// TIA Portal project "binhtron" (V15)

(* hardware
DEVICE "S7-1200 station_1"  S7-1200 Station
   slot 0: "Rack_0"  S7-1200 Rack  Rack  V1.0
   slot 1: "PLC_1"  CPU 1212C DC/DC/DC  6ES7 212-1AE40-0XB0  V4.2
DEVICE "HMI_1"  TP1500 Comfort
   slot 0: "HMI_1"  TP1500 Comfort  6AV2 124-0QC02-0AX1  15.0.0.0
   slot 1: "HMI_RT_1"  TP1500 Comfort  6AV2 124-0QC02-0AX1  15.0.0.0
   slot 5: "HMI_1.IE_CP_1"  PROFINET Interface  15.0.0.0
      slot 1: "PROFINET Interface_1"  PROFINET Interface
         slot 1: "Port_1"  Port
         slot 2: "Port_2"  Port
   slot 6: "HMI_1.IE_CP_2"  PROFINET Interface  15.0.0.0
      slot 1: "PROFINET Interface_GBit"  PROFINET Interface
         slot 1: "Port_1"  Port
   slot 7: "HMI_1.MPI/DP_CP_1"  MPI/DP Interface  15.0.0.0
*)

// ===== PLC "PLC_1"  CPU 1212C DC/DC/DC =====

VAR_GLOBAL   // PLC tag table "Default tag table"
   "System_Byte" AT %MB1 : Byte;
   "FirstScan" AT %M1.0 : Bool;
   "DiagStatusUpdate" AT %M1.1 : Bool;
   "AlwaysTRUE" AT %M1.2 : Bool;
   "AlwaysFALSE" AT %M1.3 : Bool;
   "Clock_Byte" AT %MB0 : Byte;
   "Clock_10Hz" AT %M0.0 : Bool;
   "Clock_5Hz" AT %M0.1 : Bool;
   "Clock_2.5Hz" AT %M0.2 : Bool;
   "Clock_2Hz" AT %M0.3 : Bool;
   "Clock_1.25Hz" AT %M0.4 : Bool;
   "Clock_1Hz" AT %M0.5 : Bool;
   "Clock_0.625Hz" AT %M0.6 : Bool;
   "Clock_0.5Hz" AT %M0.7 : Bool;
   "Pump" AT %Q0.0 : Bool;
   "V" AT %Q0.1 : Bool;
END_VAR

DATA_BLOCK "DB"   // DB1
{ S7_Optimized_Access := 'FALSE' }
VERSION : 0.1
   VAR
      Auto_Man : Bool;
      Start_auto : Bool;
      Stop_auto : Bool;
      Auto : Bool;
      Pump_auto : Bool;
      V_auto : Bool;
      S1_hight : Bool;
      S2_low : Bool;
      TG : Bool;
      PV_T1 : DInt;
      PV_T2 : DInt;
      start_man_pump : Bool;
      stop_man_pump : Bool;
      pump_man : Bool;
      V_man : Bool;
      start_man_V : Bool;
      stop_man_V : Bool;
      level_water : DInt;
   END_VAR
BEGIN
END_DATA_BLOCK

// folder: System blocks/Program resources

DATA_BLOCK "IEC_Timer_0_DB"   // DB2
{ S7_Optimized_Access := 'TRUE' }
AUTHOR : Simatic
FAMILY : IEC
NAME : IEC_TMR
VERSION : 1.0
// stored: InstanceOfName IEC_TIMER
"IEC_TIMER"
BEGIN
END_DATA_BLOCK

DATA_BLOCK "T2"   // DB3
{ S7_Optimized_Access := 'TRUE' }
AUTHOR : Simatic
FAMILY : IEC
NAME : IEC_TMR
VERSION : 1.0
// stored: InstanceOfName IEC_TIMER
"IEC_TIMER"
BEGIN
END_DATA_BLOCK

DATA_BLOCK "IEC_Counter_0_DB"   // DB4
{ S7_Optimized_Access := 'TRUE' }
AUTHOR : Simatic
FAMILY : IEC
NAME : CNTR
VERSION : 1.0
// stored: InstanceOfName IEC_COUNTER
"IEC_COUNTER"
BEGIN
END_DATA_BLOCK

// folder: (top level)

FUNCTION "Auto" : Void   // FC1, LAD
{ S7_Optimized_Access := 'TRUE' }
VERSION : 0.1
   VAR_TEMP   // added for the SCL form of the ladder/FBD networks
      _w1 : Bool;
   END_VAR
BEGIN

REGION Network 1
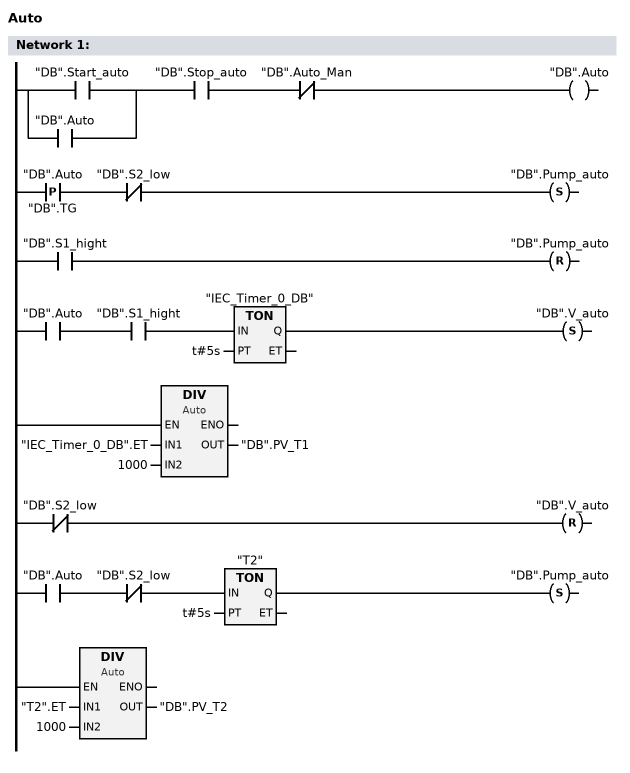
   "DB".Auto := ("DB".Start_auto OR "DB".Auto) AND "DB".Stop_auto AND NOT "DB".Auto_Man;
   #_w1 := "DB".Auto AND NOT "DB".TG;   // rising edge of "DB".Auto
   "DB".TG := "DB".Auto;
   IF #_w1 AND NOT "DB".S2_low THEN "DB".Pump_auto := TRUE; END_IF;
   IF "DB".S1_hight THEN "DB".Pump_auto := FALSE; END_IF;
   "IEC_Timer_0_DB".TON(IN := "DB".Auto AND "DB".S1_hight, PT := t#5s);
   IF "IEC_Timer_0_DB".Q THEN "DB".V_auto := TRUE; END_IF;
   "DB".PV_T1 := "IEC_Timer_0_DB".ET / 1000;
   IF NOT "DB".S2_low THEN "DB".V_auto := FALSE; END_IF;
   "T2".TON(IN := "DB".Auto AND NOT "DB".S2_low, PT := t#5s);
   IF "T2".Q THEN "DB".Pump_auto := TRUE; END_IF;
   "DB".PV_T2 := "T2".ET / 1000;
END_REGION
END_FUNCTION

FUNCTION "Man" : Void   // FC2, LAD
{ S7_Optimized_Access := 'TRUE' }
VERSION : 0.1
BEGIN

REGION Network 1
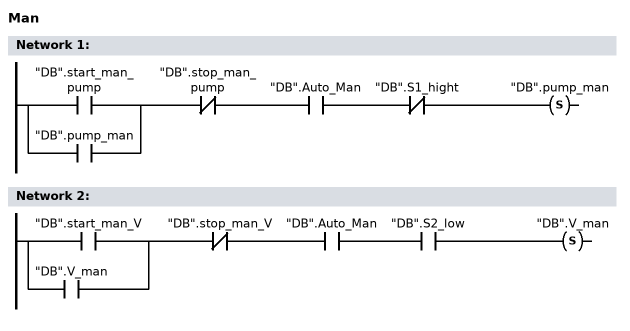
   RUNG wire#powerrail
      Contact( "DB".start_man_pump )
      wire#w1
      I_Contact( "DB".stop_man_pump )
      Contact( "DB".Auto_Man )
      I_Contact( "DB".S1_hight )
      S_Coil( "DB".pump_man )
   END_RUNG
   RUNG wire#powerrail
      Contact( "DB".pump_man )
   END_RUNG wire#w1
   // the same network as SCL:
   IF ("DB".start_man_pump OR "DB".pump_man) AND NOT "DB".stop_man_pump AND "DB".Auto_Man AND NOT "DB".S1_hight THEN
       "DB".pump_man := TRUE;
   END_IF;
END_REGION

REGION Network 2
   RUNG wire#powerrail
      Contact( "DB".start_man_V )
      wire#w1
      I_Contact( "DB".stop_man_V )
      Contact( "DB".Auto_Man )
      Contact( "DB".S2_low )
      S_Coil( "DB".V_man )
   END_RUNG
   RUNG wire#powerrail
      Contact( "DB".V_man )
   END_RUNG wire#w1
   // the same network as SCL:
   IF ("DB".start_man_V OR "DB".V_man) AND NOT "DB".stop_man_V AND "DB".Auto_Man AND "DB".S2_low THEN
       "DB".V_man := TRUE;
   END_IF;
END_REGION
END_FUNCTION

FUNCTION "Map_out" : Void   // FC3, LAD
{ S7_Optimized_Access := 'TRUE' }
VERSION : 0.1
BEGIN

REGION Network 1
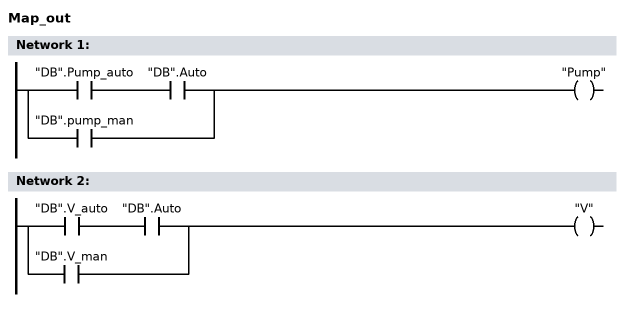
   RUNG wire#powerrail
      Contact( "DB".Pump_auto )
      Contact( "DB".Auto )
      wire#w1
      Coil( "Pump" )
   END_RUNG
   RUNG wire#powerrail
      Contact( "DB".pump_man )
   END_RUNG wire#w1
   // the same network as SCL:
   "Pump" := ("DB".Pump_auto AND "DB".Auto) OR "DB".pump_man;
END_REGION

REGION Network 2
   RUNG wire#powerrail
      Contact( "DB".V_auto )
      Contact( "DB".Auto )
      wire#w1
      Coil( "V" )
   END_RUNG
   RUNG wire#powerrail
      Contact( "DB".V_man )
   END_RUNG wire#w1
   // the same network as SCL:
   "V" := ("DB".V_auto AND "DB".Auto) OR "DB".V_man;
END_REGION
END_FUNCTION

FUNCTION "HMI_mucnuoc_sensor" : Void   // FC4, LAD
{ S7_Optimized_Access := 'TRUE' }
VERSION : 0.1
BEGIN

REGION Network 1
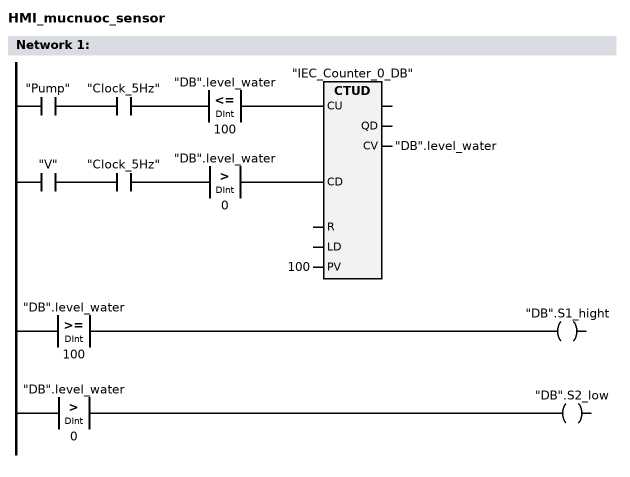
   "IEC_Counter_0_DB".CTUD(CU := "Pump" AND "Clock_5Hz" AND ("DB".level_water <= 100),
                           CD := "V" AND "Clock_5Hz" AND ("DB".level_water > 0),
                           PV := 100,
                           CV => "DB".level_water);
   "DB".S1_hight := "DB".level_water >= 100;
   "DB".S2_low := "DB".level_water > 0;
END_REGION
END_FUNCTION

ORGANIZATION_BLOCK "Main"   // OB1, LAD, ProgramCycle
TITLE = "Main Program Sweep (Cycle)"
{ S7_Optimized_Access := 'TRUE' }
VERSION : 0.1
   VAR_INPUT
      Initial_Call : Bool;   // Initial call of this OB
      Remanence : Bool;   // =True, if remanent data are available
   END_VAR
BEGIN

REGION Network 1
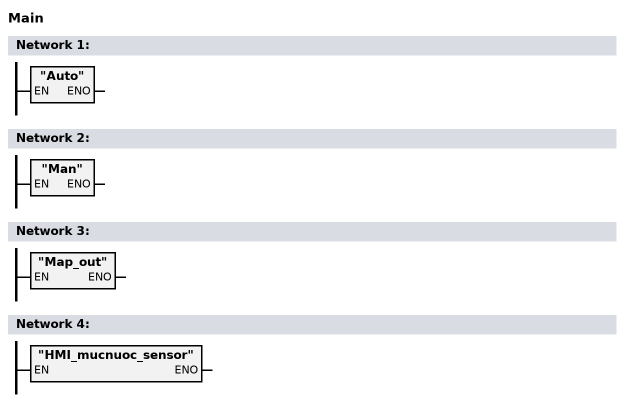
   RUNG wire#powerrail
      "Auto"()
   END_RUNG
   // the same network as SCL:
   "Auto"();
END_REGION

REGION Network 2
   RUNG wire#powerrail
      "Man"()
   END_RUNG
   // the same network as SCL:
   "Man"();
END_REGION

REGION Network 3
   RUNG wire#powerrail
      "Map_out"()
   END_RUNG
   // the same network as SCL:
   "Map_out"();
END_REGION

REGION Network 4
   RUNG wire#powerrail
      "HMI_mucnuoc_sensor"()
   END_RUNG
   // the same network as SCL:
   "HMI_mucnuoc_sensor"();
END_REGION
END_ORGANIZATION_BLOCK

(* ===== HMI "HMI_RT_1" =====
system functions are stored by id; their names below are inferred from use
connection "HMI_Connection_1": ETHERNET, S7_1200_OMS

HMI tags "Default tag table"
   "DB_Auto_Man" : Bool = PLC "DB".Auto_Man AT %DB1.DBX0.0, 1 s
   "DB_Start_auto" : Bool = PLC "DB".Start_auto AT %DB1.DBX0.1, 1 s
   "DB_Stop_auto" : Bool = PLC "DB".Stop_auto AT %DB1.DBX0.2, 1 s
   "Pump" : Bool = PLC Pump AT %Q0.0, 1 s
   "DB_level_water" : DInt = PLC "DB".level_water AT %DB1.DBD12, 1 s
   "V" : Bool = PLC V AT %Q0.1, 1 s
   "DB_S1_hight" : Bool = PLC "DB".S1_hight AT %DB1.DBX0.6, 1 s
   "DB_S2_low" : Bool = PLC "DB".S2_low AT %DB1.DBX0.7, 1 s
   "DB_PV_T1" : DInt = PLC "DB".PV_T1 AT %DB1.DBD2, 1 s
   "DB_PV_T2" : DInt = PLC "DB".PV_T2 AT %DB1.DBD6, 1 s

Template "Template_1" 1280x800
   Button "Exit" at 1200,739 size 78x59; TextOff 'Exit'; PictureOff "ExitRuntime_TP1500_Comfort_V2_TR"; PictureOn "ExitRuntime_TP1500_Comfort_V2_TR"
      on Release: StopRuntime(0)
   Button "Template_Button" at 1120,739 size 78x59; TextOff 'Text'
   Button "Template_Button_1" at 1040,739 size 78x59; TextOff 'Text'
   Button "Template_Button_2" at 960,739 size 78x59; TextOff 'Text'
   Button "Template_Button_3" at 880,739 size 78x59; TextOff 'Text'
   Button "Template_Button_4" at 800,739 size 78x59; TextOff 'Text'
   Button "Template_Button_5" at 720,739 size 78x59; TextOff 'Text'
   Button "Template_Button_6" at 640,739 size 78x59; TextOff 'Text'
   Button "Template_Button_7" at 561,739 size 78x59; TextOff 'Text'
   Button "Template_Button_8" at 481,739 size 78x59; TextOff 'Text'
   Button "Template_Button_9" at 401,739 size 78x59; TextOff 'Text'
   Button "Template_Button_10" at 321,739 size 78x59; TextOff 'Text'
   Button "Template_Button_11" at 241,739 size 78x59; TextOff 'Text'
   Button "Template_Button_12" at 161,739 size 78x59; TextOff 'Text'
   Button "Template_Button_13" at 81,739 size 78x59; TextOff 'Text'
   Button "Start screen" at 1,739 size 78x59; TextOff 'Start screen'; PictureOff "NavigateHome_TP1500_Comfort_V2_TR"; PictureOn "NavigateHome_TP1500_Comfort_V2_TR"
      on Release: ActivateScreen("Root screen", 0)

screen "Screen_1" 1280x800
   TextField "Text field_1" at 111,127 size 46x25; Text 'Text'
   TextField "Text field_2" at 80,109 size 143x29; Text 'Select mode'
   TextField "Text field_3" at 64,187 size 57x29; Text 'auto'
   TextField "Text field_4" at 184,190 size 54x29; Text 'man'
   Circle "Circle_1" at 184,144 size 48x48
      Appearance <- "DB_Auto_Man"
   Circle "Circle_2" at 63,144 size 48x48
      Appearance <- "DB_Auto_Man"
   Button "Button_1" at 104,236 size 105x49; TextOff 'Select'
   Circle "Circle_3" at 134,321 size 48x48
      Appearance <- "DB_Auto_Man"
   TextField "Text field_5" at 132,362 size 57x29; Text 'auto'
   Button "Button_2" at 106,398 size 96x32; TextOff 'Start'
      on Release: ResetBit("DB_Stop_auto")
      on Press: SetBit("DB_Start_auto")
      Appearance <- "DB_Start_auto"
   Button "Button_3" at 107,441 size 96x32; TextOff 'Stop'
      on Release: ResetBit("DB_Stop_auto")
      on Press: SetBit("DB_Stop_auto")
      Appearance <- "DB_Stop_auto"
   SymbolLibrary "Symbol library_1" at 330,416 size 222x120
      Appearance <- "Pump"
   SymbolLibrary "Symbol library_2" at 671,69 size 185x300
   Slider "Slider_1" at 673,75 size 180x239; Caption 'SIMATIC'
      ProcessValue <- "DB_level_water"
   SymbolLibrary "Symbol library_3" at 853,67 size 100x38
      Appearance <- "DB_S1_hight"
   SymbolLibrary "Symbol library_4" at 493,9 size 59x73
   SymbolLibrary "Symbol library_5" at 494,61 size 28x359
   SymbolLibrary "Symbol library_6" at 524,10 size 200x28
   SymbolLibrary "Symbol library_7" at 688,7 size 73x59
   SymbolLibrary "Symbol library_8" at 763,388 size 28x120
   SymbolLibrary "Symbol library_9" at 855,279 size 100x38
      Appearance <- "DB_S2_low"
   IOField "I/O field_1" at 1028,59 size 96x32; FormatPattern 9999999999
      Appearance <- "DB_PV_T1"
      ProcessValue <- "DB_PV_T1"
   TextField "Text field_6" at 1133,59 size 33x29; Text 'T1'
   IOField "I/O field_2" at 1027,119 size 96x32; FormatPattern 9999999999
      Appearance <- "DB_PV_T1"
      ProcessValue <- "DB_PV_T2"
   TextField "Text field_7" at 1132,119 size 33x29; Text 'T2'
   SymbolLibrary "Symbol library_10" at 710,319 size 120x72
      Appearance <- "V"
*)